TYPE ECnv_Settings_DUT :
STRUCT
	ID:	DINT;
	Barcode_ID:	UINT;
	Cnv_Level:	UINT;
	TC_Time:	UINT;
	Transfer_Time:	UINT;
	Pallet_Align_Time:	UINT;
	Slow_Speed:	UINT;
	Full_Speed:	UINT;
	Manual_Speed:	UINT;
END_STRUCT
END_TYPE

(* stored: Version 1.1.0.1
   DUT ECnv_Settings_DUT: Id {ea80fb7d-cbd2-48e1-99ad-9458c55b881e} *)
